FUNCTION_BLOCK SERVER_1_2 (* 2 RD/1 SD Server Interface *)
  (* Standard: 61499-1 *)
  (* Version 0.2, 2008-06-04, JHC, Holobloc Inc, Updated DOCTYPE. *)
  (* Version 0.1, 2001-04-25, JHC, Rockwell Automation, XML version *)
  (* Version 0.0, 1999-07-22, JHC, Rockwell Automation, SRC version *)
  (* Compiler header: package fb.rt.net; *)
  (* Compiler Java IBM VisualAge 3.0 *)
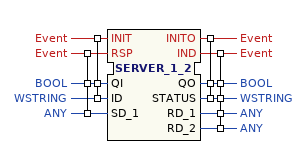
  EVENT_INPUT
    INIT WITH QI, ID; (* Service Initialization *)
    RSP WITH QI, SD_1; (* Service Response *)
  END_EVENT
  EVENT_OUTPUT
    INITO WITH QO, STATUS; (* Initialization Confirm *)
    IND WITH QO, STATUS, RD_1, RD_2; (* Service Indication *)
  END_EVENT
  VAR_INPUT
    QI : BOOL; (* Event Input Qualifier *)
    ID : WSTRING; (* Connection Identifier *)
    SD_1 : ANY; (* Data to Send *)
  END_VAR
  VAR_OUTPUT
    QO : BOOL; (* Event Output Qualifier *)
    STATUS : WSTRING; (* Service Status *)
    RD_1 : ANY; (* Received Data *)
    RD_2 : ANY; (* Received Data *)
  END_VAR
END_FUNCTION_BLOCK
